TYPE EL6910_PLCTOHW_PDOS :
	STRUCT
		
		ErrorAcknowledgement AT %Q* : BOOL;
		safetyReset AT %Q* : BOOL;
	
		Run AT %Q* : BOOL;
		
	END_STRUCT
END_TYPE

(* stored: Version 1.1.0.1, ProductVersion 3.1.4024.15
   DUT EL6910_PLCTOHW_PDOS: Id {9181818c-f3a8-40e4-bb88-ba84fbc71240} *)
